FUNCTION_BLOCK SocketConnectTask IMPLEMENTS ITask
VAR_INPUT
END_VAR
VAR_OUTPUT
END_VAR
VAR
	_execute : BOOL;
	iState: INT;
	_done: BOOL;
	_busy: BOOL;
	_error: BOOL;
	fbSocketConnect : Tc2_TcpIp.FB_SocketConnect;
END_VAR

CASE iState OF
	0:
		IF _execute THEN
			_done := FALSE;
			_busy := TRUE;
			_error := FALSE;
			fbSocketConnect.bExecute := TRUE;
			IF fbSocketConnect.bBusy THEN
				iState := 10;
				_execute := false;
			END_IF
		END_IF
	10:
		IF NOT fbSocketConnect.bBusy THEN
			IF NOT fbSocketConnect.bError THEN
				_done := TRUE;
			ELSE
				_error := TRUE;
			END_IF
			_busy := FALSE;
			fbSocketConnect.bExecute := FALSE;
			iState := 0;
		END_IF
END_CASE

fbSocketConnect(tTimeout := Tc2_System.DEFAULT_ADS_TIMEOUT);

METHOD Abort : BOOL
fbSocketConnect.bExecute := FALSE;
_busy := FALSE;
_execute := FALSE;
Abort := TRUE;
iState := 0;
END_METHOD

PROPERTY Busy : BOOL
GET
Busy := _busy;
END_GET
END_PROPERTY

PROPERTY Done : BOOL
GET
Done := _done;
END_GET
END_PROPERTY

PROPERTY Error : BOOL
GET
Error := _error;
END_GET
END_PROPERTY

METHOD Execute : BOOL
VAR_INPUT
	RemoteIPAddress : Tc2_System.T_IPv4Addr;
	RemotePortNumber : UDINT;
END_VAR
IF NOT fbSocketConnect.bBusy THEN
	fbSocketConnect.sRemoteHost := RemoteIPAddress;
	fbSocketConnect.nRemotePort := RemotePortNumber;	
	Execute := _execute := TRUE;
END_IF
END_METHOD

PROPERTY PUBLIC RemoteSocket : T_HSOCKET
GET
RemoteSocket := fbSocketConnect.hSocket;
END_GET
END_PROPERTY

END_FUNCTION_BLOCK

(* stored: Version 1.1.0.1, ProductVersion 3.1.4024.12
   POU SocketConnectTask: Id {2b70532e-27c4-4506-b229-171817f6d923}, SpecialFunc None
   Method Abort: Id {e4aa42f9-d87f-4e4b-a773-71a0fbccc200}
   Property Busy: Id {99ecb043-ed86-44ef-983b-f4d1d771397c}
   Get Get: Id {45a57b1d-bcdf-4e55-a55b-31b586c085ae}
   Property Done: Id {14989fd3-06b2-45d4-a584-531f1af8cb68}
   Get Get: Id {2898abe0-2142-45fb-9555-02cb3e211637}
   Property Error: Id {e65bb880-6e13-4735-a1f1-515626c82e29}
   Get Get: Id {e803e23e-0526-470c-90db-c41bf3d9cc0b}
   Method Execute: Id {4393e776-0714-415c-8eae-121ca1492023}
   Property RemoteSocket: Id {c858a190-ce00-4189-9ba9-b208e0d325c9}
   Get Get: Id {899f61b2-f610-47b9-b9e0-1fb6a2ec1483} *)
